SUBAPPLICATION Uebung_010e_PC_A_OPC (* Geraet A (Station 11, 192.168.1.11): 3 SoftKeys (Set/Reset/Toggle) rufen je einen eigenen argument- und rueckgabewertlosen OPC-UA-Methodenaufruf auf Geraet B auf (CLIENT_0, 3 eigene Methoden statt 1 String-Parameter - Option A); GreenWhiteBackground am Toggle-SoftKey zeigt den von Geraet B lokal ueberwachten Flipflop-Zustand - 'SUB style': das Protokoll steckt im MyLib::sys-Composite, nicht in der Resource des Geraets *)
  (* Standard: 61499-2; Description: Copyright (c) 2026 Meisterschulen am Ostbahnhof This program and the accompanying materials are made available under the terms of the Eclipse Public License 2.0 which is available at https://www.eclipse.org/legal/epl-2.0/ SPDX-License-Identifier: EPL-2.0 *)
  (* Version 1.0, 2026-09-02, Franz Höpfinger, Meisterschulen am Ostbahnhof, initial API and implementation and/or initial documentation *)
  PACKAGE MyLib::sys;
  IMPORT isobus::UT::Q::const::IDs::ID_NULL;
  IMPORT isobus::UT::io::Softkey::SoftKeyActivationCode::SK_RELEASED;
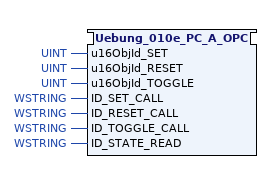
  VAR_INPUT
    u16ObjId_SET : UINT := ID_NULL; (* Object ID SoftKey Set *)
    u16ObjId_RESET : UINT := ID_NULL; (* Object ID SoftKey Reset *)
    u16ObjId_TOGGLE : UINT := ID_NULL; (* Object ID SoftKey Toggle (traegt auch das GreenWhiteBackground) *)
    ID_SET_CALL : WSTRING; (* Remote-Methodenadresse (ACTION=CALL_METHOD) fuer den Set-Methodenaufruf auf Geraet B *)
    ID_RESET_CALL : WSTRING; (* Remote-Methodenadresse (ACTION=CALL_METHOD) fuer den Reset-Methodenaufruf auf Geraet B *)
    ID_TOGGLE_CALL : WSTRING; (* Remote-Methodenadresse (ACTION=CALL_METHOD) fuer den Toggle-Methodenaufruf auf Geraet B *)
    ID_STATE_READ : WSTRING; (* Lokal ueberwachte Adresse (BOOL, ACTION=READ) fuer den Flipflop-Zustand, wird von Geraet B remote beschrieben *)
  END_VAR
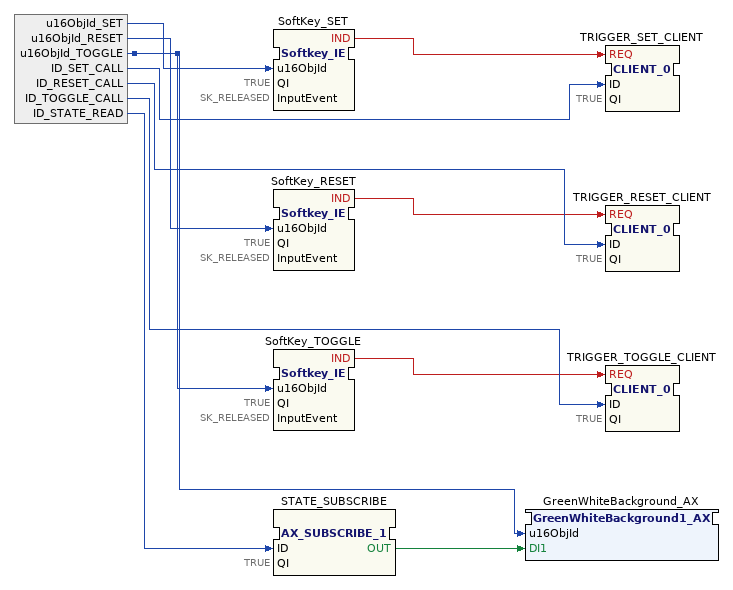
  FBS
    SoftKey_SET : isobus::UT::io::Softkey::Softkey_IE(QI := TRUE, InputEvent := SK_RELEASED);
    SoftKey_RESET : isobus::UT::io::Softkey::Softkey_IE(QI := TRUE, InputEvent := SK_RELEASED);
    SoftKey_TOGGLE : isobus::UT::io::Softkey::Softkey_IE(QI := TRUE, InputEvent := SK_RELEASED);
    TRIGGER_SET_CLIENT : iec61499::net::CLIENT_0(QI := TRUE);
    TRIGGER_RESET_CLIENT : iec61499::net::CLIENT_0(QI := TRUE);
    TRIGGER_TOGGLE_CLIENT : iec61499::net::CLIENT_0(QI := TRUE);
    STATE_SUBSCRIBE : adapter::net::AX_SUBSCRIBE_1(QI := TRUE);
  END_FBS
  SUBAPPS
    GreenWhiteBackground_AX : MyLib::sys::GreenWhiteBackground1_AX;
  END_SUBAPPS
  EVENT_CONNECTIONS
    SoftKey_SET.IND TO TRIGGER_SET_CLIENT.REQ;
    SoftKey_RESET.IND TO TRIGGER_RESET_CLIENT.REQ;
    SoftKey_TOGGLE.IND TO TRIGGER_TOGGLE_CLIENT.REQ;
  END_CONNECTIONS
  DATA_CONNECTIONS
    u16ObjId_SET TO SoftKey_SET.u16ObjId;
    u16ObjId_RESET TO SoftKey_RESET.u16ObjId;
    u16ObjId_TOGGLE TO SoftKey_TOGGLE.u16ObjId;
    u16ObjId_TOGGLE TO GreenWhiteBackground_AX.u16ObjId;
    ID_SET_CALL TO TRIGGER_SET_CLIENT.ID;
    ID_RESET_CALL TO TRIGGER_RESET_CLIENT.ID;
    ID_TOGGLE_CALL TO TRIGGER_TOGGLE_CLIENT.ID;
    ID_STATE_READ TO STATE_SUBSCRIBE.ID;
  END_CONNECTIONS
  ADAPTER_CONNECTIONS
    STATE_SUBSCRIBE.OUT TO GreenWhiteBackground_AX.DI1;
  END_CONNECTIONS
END_SUBAPPLICATION
